Yaskawa INFORM job: OK_R2_O27-28(-60,-90)OKKR.JBI

/JOB
//NAME OK_R2_O27-28(-60,-90)OKKR
///FOLDERNAME X4
//POS
///NPOS 259,259,259,8,0,0
///TOOL 0
///POSTYPE PULSE
///PULSE
C00000=4026,-114538,-112087,-7469,89169,3010
C00001=141886,-58901,-77773,-23947,92184,48931
C00002=141578,-57959,-69842,-23828,88059,49648
C00003=141015,-58362,-68930,-23729,87194,49620
C00004=141015,-58433,-67903,-23734,86579,49742
C00005=141015,-58416,-68203,-23732,86757,49707
C00006=139686,-59077,-68559,-23492,86274,49323
C00007=141015,-58416,-68203,-23732,86757,49707
C00008=141015,-58175,-70675,-23724,88270,49406
C00009=128422,-62662,-73061,-21186,84142,45699
C00010=126942,-63006,-72152,-20876,83082,45360
C00011=125859,-63161,-72230,-20632,82787,45027
C00012=126427,-63083,-72191,-20760,82941,45202
C00013=126427,-63151,-70840,-20793,82126,45342
C00014=126555,-60703,-71087,-20771,83482,45154
C00015=126555,-60807,-69619,-20804,82583,45308
C00016=127911,-60340,-72276,-21054,84679,45425
C00017=126649,-37475,-64724,-20742,91025,43893
C00018=125827,-36059,-63222,-20543,90649,43679
C00019=125029,-36163,-63287,-20349,90451,43443
C00020=125623,-36090,-63238,-20492,90597,43620
C00021=125567,-34509,-61579,-20475,90388,43635
C00022=125623,-36090,-63238,-20492,90597,43620
C00023=136338,-54772,-80020,-22951,93924,46664
C00024=126842,-100836,-98035,7484,62353,-34456
C00025=121554,-58479,-70523,23610,81393,-54658
C00026=122608,-55102,-66306,23365,80313,-54492
C00027=122608,-55177,-65231,23407,79671,-54618
C00028=122608,-55168,-65391,23401,79766,-54599
C00029=123914,-55086,-65345,23053,79422,-54193
C00030=122608,-54831,-68633,23286,81762,-54205
C00031=135057,-52399,-66134,19707,78324,-50392
C00032=136320,-52036,-64863,19353,77466,-50085
C00033=137087,-51720,-64683,19108,77338,-49833
C00034=136456,-51981,-64832,19310,77443,-50041
C00035=136456,-52079,-63836,19355,76815,-50143
C00036=136990,-51767,-64649,19142,77318,-49872
C00037=137022,-51845,-63710,19174,76726,-49958
C00038=136456,-51987,-64775,19313,77407,-50047
C00039=133944,-28024,-57248,19775,85241,-49647
C00040=134132,-26753,-56119,19717,85158,-49597
C00041=134834,-26485,-55932,19497,85022,-49384
C00042=134200,-26728,-56101,19696,85144,-49576
C00043=134114,-25902,-54940,19729,84890,-49647
C00044=134200,-26728,-56101,19696,85144,-49576
C00045=118482,-33028,-63104,24263,90056,-53997
C00046=122367,-92922,-80640,24281,48069,-47816
C00047=126786,-89890,-74695,22151,44886,-46448
C00048=127161,-97737,-79785,22235,43950,-46500
C00049=123248,-90194,-74818,24549,45815,-47997
C00050=127415,-97816,-73172,23855,40088,-47458
C00051=126170,-63328,-70330,17365,77748,-40778
C00052=125190,-29892,-53752,19424,104543,-36953
C00053=126048,-60244,-72015,19024,100224,-37353
C00054=129257,-118219,-89475,18745,55248,-43183
C00055=137691,-142606,-72024,68262,8176,-68089
C00056=133583,-154957,-83359,69355,10840,-69277
C00057=143208,-69932,-76566,3835,55131,-38143
C00058=145269,-69372,-74031,2532,53783,-37349
C00059=145623,-70560,-74318,2309,53334,-37215
C00060=145877,-71977,-74674,2159,52821,-37126
C00061=150479,-88391,-71295,-7827,30676,-34231
C00062=155149,-99562,-68728,-17073,24216,-29422
C00063=155171,-99618,-68748,-17116,24204,-29400
C00064=147593,-80029,-75214,3987,58057,-35963
C00065=135411,-30256,-54215,19906,99237,-39191
C00066=136924,-45266,-63867,20529,99583,-42128
C00067=135919,-63282,-79199,18518,95221,-35974
C00068=132995,-62152,-82050,19008,98077,-36535
C00069=146597,-77867,-86304,-14777,77362,40583
C00070=149051,-83920,-77966,-27962,61330,43366
C00071=147016,-82878,-78861,-27270,61762,42356
C00072=150258,-80090,-74192,-28972,61572,43794
C00073=147203,-82736,-75214,-27895,59886,42937
C00074=149174,-90821,-74362,-30094,56451,44819
C00075=149181,-90838,-74335,-30106,56432,44829
C00076=142127,-55357,-68668,-16008,88190,36417
C00077=139597,-29306,-55135,-13561,105265,43860
C00078=139307,-22183,-50052,-13420,110648,48850
C00079=143000,-50940,-68567,-12955,107923,50473
C00080=151384,-106281,-89249,-20779,70795,55648
C00081=160066,-126367,-88243,-34868,53700,64122
C00082=163396,-129603,-85950,-37116,52558,66246
C00083=170124,-141759,-99198,-37878,56949,67763
C00084=136065,-86573,-88427,-19738,64261,50781
C00085=131238,-34371,-67556,-16142,92767,44746
C00086=129250,-31705,-63617,-15587,92385,44136
C00087=129352,-32707,-64477,-15613,92413,44167
C00088=131697,-69478,-76768,-20363,65108,48613
C00089=131773,-70326,-76955,-20450,64822,48696
C00090=132058,-74122,-77463,-20852,63359,49080
C00091=133339,-88291,-77768,-22923,57086,50905
C00092=133349,-88399,-77812,-22935,57064,50915
C00093=131196,-63810,-72799,-16490,80948,46201
C00094=129177,-28734,-55041,-14328,108045,42506
C00095=130098,-48812,-67542,-14099,105651,43119
C00096=135207,-44513,-73407,-14614,112147,44115
C00097=29949,-45667,-74098,-14599,111934,44036
C00098=58439,-77793,-131196,12526,65130,-72907
C00099=127967,-68734,-129505,14303,77633,-40887
C00100=95610,-66837,-124865,12878,106964,29326
C00101=114477,-82986,-128069,-10037,99362,30876
C00102=114477,-86675,-127599,-9968,97208,31049
C00103=114477,-85869,-127717,-9982,97688,31010
C00104=112971,-85457,-127558,-9480,97652,30583
C00105=92898,-68043,-124184,12345,107279,29217
C00106=94676,-96172,-135168,11342,99536,28957
C00107=94658,-98853,-133311,11256,97065,28724
C00108=95162,-93948,-131570,11149,98431,28996
C00109=94658,-98853,-133311,11256,97065,28724
C00110=98957,-93279,-135892,10098,100972,30314
C00111=110651,-49645,-111382,-11454,101977,41926
C00112=110651,-52306,-111062,-11381,100444,42072
C00113=110651,-51032,-111225,-11415,101184,42001
C00114=109332,-50612,-111005,-10903,101130,41666
C00115=110651,-51032,-111225,-11415,101184,42001
C00116=95349,-81608,-124870,6979,89211,41800
C00117=95569,-84274,-123262,6885,86851,41730
C00118=95987,-80853,-121877,6703,87721,41895
C00119=95620,-84218,-124899,6861,87878,41800
C00120=95569,-64927,-125294,6988,97966,42345
C00121=68892,-69920,-123147,37382,97488,27376
C00122=68892,-69920,-123147,37382,97488,27376
C00123=68031,-90449,-131916,26273,102698,-13010
C00124=71990,-90821,-130319,24971,100628,-12221
C00125=79202,-85723,-129933,18399,102227,-11158
C00126=79202,-87573,-129743,18299,101214,-11319
C00127=79215,-86748,-129802,18348,101647,-11244
C00128=80019,-82599,-128205,18192,102594,-10863
C00129=79215,-83561,-130075,18500,103364,-10977
C00130=72693,-92471,-130926,24716,100020,-12130
C00131=84462,-79485,-128908,14471,105620,-10048
C00132=84462,-81364,-128782,14389,104604,-10171
C00133=84462,-80152,-128866,14442,105265,-10090
C00134=85127,-76283,-127309,14327,106169,-9791
C00135=84083,-80509,-129856,14589,105729,-10142
C00136=72693,-92471,-130926,24716,100020,-12130
C00137=84410,-93585,-133880,14135,99565,-10800
C00138=84410,-96087,-133656,14067,98184,-10958
C00139=84410,-94757,-133784,14102,98923,-10874
C00140=85385,-88254,-131421,13878,100620,-10395
C00141=84410,-93524,-133885,14136,99597,-10796
C00142=71593,-80403,-130713,25764,105804,-11193
C00143=71593,-76518,-130795,32588,107642,-50773
C00144=78737,-74748,-122692,29451,101785,-50195
C00145=78737,-75119,-122640,29424,101590,-50246
C00146=78737,-77656,-122235,29243,100229,-50601
C00147=78737,-76000,-122510,29360,101124,-50368
C00148=80423,-78738,-123652,28717,100035,-50114
C00149=74556,-86649,-127298,30428,100128,-51983
C00150=80828,-115772,-134875,23515,87622,-34169
C00151=81779,-109674,-132899,23210,89145,-33553
C00152=81251,-111521,-134487,23382,89304,-33698
C00153=81251,-105171,-135824,23470,93068,-32958
C00154=68840,-107115,-136272,27319,95724,-36434
C00155=63225,-73448,-121715,35441,110616,-40683
C00156=63225,-75726,-121350,35103,109465,-41078
C00157=63225,-74780,-121511,35242,109948,-40913
C00158=64274,-77370,-122606,34819,109058,-40843
C00159=63225,-72176,-121887,35634,111241,-40463
C00160=49970,-81546,-125790,38107,113825,-44363
///LIMIT ON
C00161=57709,-122397,-137101,29737,92456,-40867
///LIMIT OFF
C00162=58596,-119094,-136084,29567,93103,-40381
///LIMIT ON
C00163=57709,-122397,-137101,29737,92456,-40867
///LIMIT OFF
C00164=55203,-68367,-119401,40200,117926,-44687
C00165=60082,-69241,-118655,38808,115482,-43833
C00166=70586,-91755,-127960,28719,99346,-36878
C00167=58188,-109460,-135678,31383,99168,-40913
C00168=58490,-112528,-136667,30978,97870,1529
C00169=60906,-115834,-135191,27280,87192,7891
C00170=59523,-104900,-131558,29509,92292,6762
C00171=56755,-69637,-113373,48283,106573,15620
C00172=54350,-66602,-110106,52807,107764,16888
C00173=41617,-83627,-112954,60214,104174,10782
C00174=28595,-74588,-109030,64073,112578,9715
C00175=27901,-74856,-109516,64304,113044,9684
C00176=47677,-91044,-131006,33540,104945,-26933
///LIMIT ON
C00177=61912,-123095,-136997,21835,82960,-21144
///LIMIT OFF
C00178=55245,-67359,-115879,41246,114826,-18847
C00179=56373,-63948,-120424,31486,113982,-21878
C00180=60160,-119068,-134198,40501,98040,-56836
C00181=60160,-114231,-136050,40991,100824,-55736
C00182=83270,-65163,-115072,44519,104941,-68495
C00183=85626,-71751,-115611,43145,101762,-69006
C00184=84703,-74765,-113322,46278,99950,-69048
C00185=88262,-57949,-105339,45732,101061,-67072
C00186=101128,-54439,-109788,29647,101331,-67085
C00187=94109,-71359,-120991,32482,95089,-70619
C00188=139920,-94168,-131864,-18457,87392,-68872
C00189=164516,-97279,-127794,-42983,94890,-67354
C00190=173049,-108773,-127338,-48480,95293,-64880
C00191=167455,-99667,-123526,-46768,91665,-65667
C00192=150655,-112829,-124924,-46404,81551,-69570
C00193=121485,-77048,-127419,1615,96838,-70506
C00194=141399,-68559,-121452,-18612,100542,-82408
C00195=124764,-66998,-122517,455,101591,-69580
C00196=125438,-65497,-122047,206,102070,-69406
C00197=126763,-65065,-121637,-284,102041,-69063
C00198=120566,-81356,-130422,1967,92166,-70821
C00199=120566,-76874,-130556,1975,94549,-70784
C00200=125831,-89175,-135984,-584,100456,3377
C00201=135444,-90328,-133818,-3844,98745,6043
C00202=135106,-91582,-131067,-3703,96397,6020
C00203=109572,-93250,-131605,4930,96041,-1221
C00204=87998,-80897,-129766,12221,103039,-6801
C00205=120367,-85836,-132161,9477,101125,-4686
C00206=121843,-84446,-127481,8917,98851,-4443
C00207=141527,-76678,-124327,2331,99777,1071
C00208=129396,-87762,-136435,6506,102049,-2146
C00209=130312,-90929,-132015,6094,97669,-2118
C00210=129363,-86126,-129166,6424,98441,-2343
C00211=154391,-66262,-120817,-2111,102954,4533
C00212=150219,-78004,-128736,-656,101737,3438
C00213=144801,-93164,-134458,-6692,98136,8453
C00214=144714,-84238,-128290,-6682,98918,8387
C00215=123987,-96369,-132727,351,94749,2642
C00216=117273,-90923,-135342,2652,99260,807
C00217=121768,-81824,-133505,6628,103406,-2316
C00218=156634,-61907,-126378,-3075,94108,-72042
C00219=137751,-95208,-134275,-20772,87240,-85897
C00220=160150,-96114,-119425,-47944,88000,-84014
C00221=155632,-76142,-111175,-46420,89477,-86695
C00222=140577,-51697,-109067,-28499,100390,-90208
C00223=132515,-86588,-130828,-12209,89399,-86569
C00224=131433,-65917,-122271,-11801,94519,-87353
C00225=105014,-130347,-135310,35662,68949,-87927
C00226=104111,-122678,-131012,37838,71563,-88295
C00227=106068,-95108,-121457,35727,77495,-85456
C00228=111976,-92342,-121116,28689,76109,-84990
C00229=109886,-91804,-124961,29447,79067,-84948
C00230=149255,-76965,-128804,-12913,97351,-82067
C00231=139576,-84817,-129459,-1876,92119,-81977
C00232=148153,-75159,-124875,-14582,97706,-83124
C00233=147471,-74687,-124680,-14327,97728,-83315
C00234=146233,-76138,-125285,-13834,97200,-83595
C00235=149105,-93032,-135747,-12738,93444,-81701
C00236=185390,-49383,-101810,-59538,112858,-87685
C00237=178512,-86634,-117153,-49673,98332,-85874
C00238=173349,-72532,-111075,-48613,98244,-88135
C00239=168036,-108473,-125463,-40279,80417,-90424
C00240=177281,-105060,-127213,-43325,86617,-89102
C00241=179538,-98194,-126909,-44097,90073,-89650
C00242=186838,-121222,-134600,-46262,88364,-34815
C00243=184942,-111108,-129526,-47770,92446,-34323
C00244=190696,-133181,-128203,-55352,82590,-27191
C00245=183298,-110716,-114958,-62940,86926,-24714
C00246=183340,-79337,-102682,-66907,100105,-26093
C00247=185184,-79882,-104966,-67590,101694,-26340
C00248=200556,-111348,-116827,-65901,96352,-23239
C00249=198058,-141281,-124059,-63896,81460,-21046
C00250=197686,-130606,-120716,-64143,86176,-21704
C00251=190742,-91685,-107319,-68355,104344,-23733
C00252=191763,-88052,-108908,-69399,106084,-24879
C00253=198707,-113921,-124746,-62747,95061,-23584
C00254=198707,-113921,-124746,-62747,95061,-23584
C00255=177230,-52335,-122859,-28636,110825,-71925
C00256=181545,-112898,-119475,-62736,95065,-23495
C00257=7977,-118181,-126139,1257,90741,84078
C00258=4441,-114902,-113556,-6551,89340,11522
BC00000=154724,492605,1071101
BC00001=345701,440224,1074748
BC00002=345701,440224,1074748
BC00003=345701,440224,1074748
BC00004=345701,440224,1074748
BC00005=345701,440224,1074748
BC00006=345701,440224,1074748
BC00007=345701,440224,1074748
BC00008=345701,440224,1074748
BC00009=345701,440224,1074748
BC00010=345701,440224,1074748
BC00011=345701,440224,1074748
BC00012=345701,440224,1074748
BC00013=345701,440224,1074748
BC00014=345701,440224,1074748
BC00015=345701,440224,1074748
BC00016=345701,440224,1074748
BC00017=345701,440224,1074748
BC00018=345701,440224,1074748
BC00019=345701,440224,1074748
BC00020=345701,440224,1074748
BC00021=345701,440224,1074748
BC00022=345701,440224,1074748
BC00023=345701,440224,1074748
BC00024=136420,445856,1074364
BC00025=136420,445856,1074364
BC00026=136419,445855,1074361
BC00027=136419,445855,1074361
BC00028=136419,445855,1074361
BC00029=136419,445855,1074361
BC00030=136419,445855,1074361
BC00031=136419,445855,1074361
BC00032=136419,445855,1074361
BC00033=136419,445855,1074361
BC00034=136419,445855,1074361
BC00035=136419,445855,1074361
BC00036=136419,445855,1074361
BC00037=136419,445855,1074361
BC00038=136419,445855,1074361
BC00039=136419,445855,1074361
BC00040=136419,445855,1074361
BC00041=136419,445855,1074361
BC00042=136419,445855,1074361
BC00043=136419,445855,1074361
BC00044=136419,445855,1074361
BC00045=136419,445855,1074361
BC00046=132124,434884,1075130
BC00047=132124,434884,1075130
BC00048=132124,434884,1075130
BC00049=132124,434884,1075130
BC00050=132125,434884,1075124
BC00051=132124,434884,1075127
BC00052=132124,434884,1075127
BC00053=132124,434884,1075127
BC00054=132124,434884,1075127
BC00055=132124,434884,1075127
BC00056=132124,434884,1075123
BC00057=132124,434884,1075123
BC00058=132124,434884,1075123
BC00059=132124,434884,1075123
BC00060=132124,434884,1075123
BC00061=132124,434884,1075123
BC00062=132124,434884,1075120
BC00063=132124,434884,1075120
BC00064=132124,434884,1075123
BC00065=132124,434884,1075120
BC00066=132124,434884,1075120
BC00067=132124,434884,1075120
BC00068=132124,434884,1075120
BC00069=365171,434884,1075120
BC00070=365171,434884,1075120
BC00071=365171,434884,1075120
BC00072=365171,434884,1075120
BC00073=365171,434884,1075120
BC00074=365171,434884,1075120
BC00075=365171,434884,1075120
BC00076=365171,434884,1075120
BC00077=365171,434884,1075120
BC00078=365171,434884,1075120
BC00079=365171,434884,1075120
BC00080=365171,434884,1075120
BC00081=365171,434884,1075120
BC00082=365171,434884,1075120
BC00083=365171,434884,1075120
BC00084=365171,434884,1075120
BC00085=365171,434884,1075120
BC00086=365171,434884,1075120
BC00087=365171,434884,1075120
BC00088=365171,434884,1075120
BC00089=365171,434884,1075120
BC00090=365171,434884,1075120
BC00091=365171,434884,1075120
BC00092=365171,434884,1075120
BC00093=365171,434884,1075120
BC00094=365171,434884,1075120
BC00095=365171,434884,1075120
BC00096=365171,434884,1075120
BC00097=261029,496377,1070955
BC00098=158954,465505,1070842
BC00099=76268,391428,1075124
BC00100=6523,355122,1075124
BC00101=1090,352294,1075124
BC00102=1090,352294,1075124
BC00103=1090,352294,1075124
BC00104=1090,352294,1075124
BC00105=1090,352294,1075124
BC00106=1090,352294,1075124
BC00107=1090,352294,1075124
BC00108=1090,352294,1075124
BC00109=1090,352294,1075124
BC00110=1090,352294,1075124
BC00111=1090,352294,1075124
BC00112=1090,352294,1075124
BC00113=1090,352294,1075124
BC00114=1090,352294,1075124
BC00115=1090,352294,1075124
BC00116=1090,352294,1075124
BC00117=1090,352294,1075124
BC00118=1090,352294,1075124
BC00119=1090,352294,1075124
BC00120=1090,352294,1075124
BC00121=1090,352294,1075124
BC00122=1090,352294,1075124
BC00123=119522,336763,1061257
BC00124=119522,336763,1061257
BC00125=119522,336763,1061257
BC00126=119523,336764,1061256
BC00127=119522,336763,1061257
BC00128=119522,336763,1061257
BC00129=119522,336763,1061257
BC00130=177823,336763,1064589
BC00131=177823,336763,1061257
BC00132=177823,336763,1061257
BC00133=177823,336763,1061257
BC00134=177823,336763,1061257
BC00135=177823,336763,1061257
BC00136=233759,336763,1064589
BC00137=233759,336315,1058464
BC00138=233759,336315,1058464
BC00139=233759,336315,1058464
BC00140=233758,336315,1058463
BC00141=233759,336315,1058464
BC00142=233759,336315,1059003
BC00143=363339,336315,1059003
BC00144=363339,336315,1059003
BC00145=363339,336315,1059003
BC00146=363339,336315,1059003
BC00147=363339,336315,1059003
BC00148=363339,336315,1059003
BC00149=363339,336315,1059003
BC00150=363339,336315,1059003
BC00151=363339,336315,1059003
BC00152=363339,336315,1059003
BC00153=363339,336315,1059003
BC00154=362736,339076,1059003
BC00155=362465,340315,1059003
BC00156=362465,340315,1059003
BC00157=362465,340315,1059003
BC00158=362465,340315,1059003
BC00159=362465,340315,1059003
BC00160=362465,340315,1059003
BC00161=362465,340315,1059003
BC00162=362465,340315,1059003
BC00163=362465,340315,1059003
BC00164=362465,340315,1059003
BC00165=362465,340315,1059003
BC00166=362465,340315,1059003
BC00167=362465,340315,1059003
BC00168=362466,340316,1059002
BC00169=349813,347319,1059002
BC00170=349813,347319,1059002
BC00171=349813,347319,1059002
BC00172=349813,347319,1059002
BC00173=349813,347319,1059002
BC00174=349813,347319,1059002
BC00175=349813,347319,1059002
BC00176=349813,347319,1059002
BC00177=348803,347319,1059002
BC00178=349813,347319,1059002
BC00179=349813,347319,1059002
BC00180=381408,339179,1066112
BC00181=381408,339179,1066112
BC00182=396370,339179,1066112
BC00183=396370,339179,1066112
BC00184=396370,339179,1066112
BC00185=396370,339179,1066112
BC00186=396370,339179,1066112
BC00187=396370,339179,1066112
BC00188=396370,330317,1066112
BC00189=396370,323887,1066112
BC00190=396370,323887,1066112
BC00191=396370,323887,1066112
BC00192=366417,324055,1066112
BC00193=396370,328332,1066112
BC00194=396370,328332,1066109
BC00195=396370,328332,1066112
BC00196=396370,328332,1066112
BC00197=396370,328332,1066112
BC00198=396370,328332,1066112
BC00199=396370,328332,1066112
BC00200=237361,342916,1066112
BC00201=237361,342915,1066109
BC00202=237361,342915,1066109
BC00203=237361,342915,1066109
BC00204=237361,342915,1066109
BC00205=204586,344800,1071989
BC00206=204586,344800,1071989
BC00207=204586,344800,1071989
BC00208=248457,342915,1066109
BC00209=248457,342915,1066109
BC00210=248457,342915,1066109
BC00211=248457,342915,1066109
BC00212=248457,342915,1066109
BC00213=280970,342915,1066109
BC00214=280970,342915,1066109
BC00215=280970,342915,1066109
BC00216=280970,342915,1066109
BC00217=250684,342915,1066109
BC00218=120387,342915,1066109
BC00219=43564,342915,1066109
BC00220=43564,342915,1066109
BC00221=43564,342915,1066109
BC00222=43564,342915,1066109
BC00223=43563,342915,1066106
BC00224=43563,352075,1066106
BC00225=77352,343027,1066106
BC00226=77352,343027,1066106
BC00227=77352,343027,1066106
BC00228=77352,343027,1066106
BC00229=77352,343027,1066106
BC00230=77352,325808,1066106
BC00231=77351,325808,1066103
BC00232=77352,325808,1066106
BC00233=77352,325808,1066106
BC00234=77352,325808,1066106
BC00235=77352,325808,1066106
BC00236=58352,353191,1066106
BC00237=58352,353191,1066106
BC00238=58352,353191,1066106
BC00239=58352,353191,1066106
BC00240=58352,353191,1066106
BC00241=58352,353191,1066106
BC00242=58352,353191,1066106
BC00243=58352,353191,1066106
BC00244=58352,353191,1066106
BC00245=58352,353191,1066106
BC00246=58352,353191,1066106
BC00247=58352,353191,1066106
BC00248=58352,353191,1066106
BC00249=58352,353191,1066106
BC00250=58352,353191,1066106
BC00251=58352,353191,1066106
BC00252=58352,353191,1066106
BC00253=58352,353191,1066106
BC00254=12917,447675,1066106
BC00255=70552,358579,1066106
BC00256=12917,447675,1066106
BC00257=12917,516869,1066106
BC00258=138844,495152,1070575
EC00000=454111,372643
EC00001=443859,372643
EC00002=443859,372643
EC00003=443859,372643
EC00004=443859,372643
EC00005=443859,372643
EC00006=443859,372643
EC00007=443859,372643
EC00008=443859,372643
EC00009=443859,372643
EC00010=443859,372643
EC00011=443859,372643
EC00012=443859,372643
EC00013=443859,372643
EC00014=443859,372643
EC00015=443859,372643
EC00016=443859,372643
EC00017=443859,372643
EC00018=443859,372643
EC00019=443859,372643
EC00020=443859,372643
EC00021=443859,372643
EC00022=443859,372643
EC00023=443859,372643
EC00024=444967,372643
EC00025=444967,372643
EC00026=444965,372643
EC00027=444965,372643
EC00028=444965,372643
EC00029=444965,372643
EC00030=444965,372643
EC00031=444965,372643
EC00032=444965,372643
EC00033=444965,372643
EC00034=444965,372643
EC00035=444965,372643
EC00036=444965,372643
EC00037=444965,372643
EC00038=444965,372643
EC00039=444965,372643
EC00040=444965,372643
EC00041=444965,372643
EC00042=444965,372643
EC00043=444965,372643
EC00044=444965,372643
EC00045=444965,372643
EC00046=442821,372643
EC00047=442821,372643
EC00048=442821,372643
EC00049=442821,372643
EC00050=442817,372643
EC00051=442818,372643
EC00052=442818,372643
EC00053=442818,372643
EC00054=442818,372643
EC00055=442818,372643
EC00056=442816,372643
EC00057=442816,372643
EC00058=442816,372643
EC00059=442816,372643
EC00060=442816,372643
EC00061=442816,372643
EC00062=442815,372643
EC00063=442815,372643
EC00064=442816,372643
EC00065=442814,372643
EC00066=442814,372643
EC00067=442814,372643
EC00068=442814,372643
EC00069=442814,372643
EC00070=442814,372643
EC00071=442814,372643
EC00072=442814,372643
EC00073=442814,372643
EC00074=442814,372643
EC00075=442814,372643
EC00076=442814,372643
EC00077=442814,372643
EC00078=442814,372643
EC00079=442814,372643
EC00080=442814,372643
EC00081=442814,372643
EC00082=442814,372643
EC00083=442814,372643
EC00084=442814,372643
EC00085=442814,372643
EC00086=442814,372643
EC00087=442814,372643
EC00088=442814,372643
EC00089=442814,372643
EC00090=442814,372643
EC00091=442814,372643
EC00092=442814,372643
EC00093=442814,372643
EC00094=442814,372643
EC00095=442814,372643
EC00096=442814,372643
EC00097=442814,372643
EC00098=798155,372644
EC00099=798157,372644
EC00100=798157,372644
EC00101=798157,372644
EC00102=798157,372644
EC00103=798157,372644
EC00104=798157,372644
EC00105=798157,372644
EC00106=798157,372644
EC00107=798157,372644
EC00108=798157,372644
EC00109=798157,372644
EC00110=798157,372644
EC00111=798157,372644
EC00112=798157,372644
EC00113=798157,372644
EC00114=798157,372644
EC00115=798157,372644
EC00116=798157,372644
EC00117=798157,372644
EC00118=798157,372644
EC00119=798157,372644
EC00120=798157,372644
EC00121=798157,372644
EC00122=798157,372644
EC00123=798157,372644
EC00124=798157,372644
EC00125=798157,372644
EC00126=798156,372644
EC00127=798157,372644
EC00128=798157,372644
EC00129=798157,372644
EC00130=798157,372644
EC00131=798157,372644
EC00132=798157,372644
EC00133=798157,372644
EC00134=798157,372644
EC00135=798157,372644
EC00136=798157,372644
EC00137=798157,372644
EC00138=798157,372644
EC00139=798157,372644
EC00140=798155,372644
EC00141=798157,372644
EC00142=798157,372644
EC00143=798157,372644
EC00144=798157,372644
EC00145=798157,372644
EC00146=798157,372644
EC00147=798157,372644
EC00148=798157,372644
EC00149=798157,372644
EC00150=798157,372644
EC00151=798157,372644
EC00152=798157,372644
EC00153=798157,372644
EC00154=798157,372644
EC00155=798157,372644
EC00156=798157,372644
EC00157=798157,372644
EC00158=798157,372644
EC00159=798157,372644
EC00160=798157,372644
EC00161=798157,372644
EC00162=798157,372644
EC00163=798157,372644
EC00164=798157,372644
EC00165=798157,372644
EC00166=798157,372644
EC00167=798157,372644
EC00168=798156,372644
EC00169=798156,372644
EC00170=798156,372644
EC00171=798156,372644
EC00172=798156,372644
EC00173=798156,372644
EC00174=798156,372644
EC00175=798156,372644
EC00176=798156,372644
EC00177=798156,372644
EC00178=798156,372644
EC00179=798156,372644
EC00180=798156,372644
EC00181=798156,372644
EC00182=798156,372644
EC00183=798156,372644
EC00184=798156,372644
EC00185=798156,372644
EC00186=798156,372644
EC00187=798156,372644
EC00188=798156,372644
EC00189=798156,372644
EC00190=798156,372644
EC00191=798156,372644
EC00192=798156,372644
EC00193=798156,372644
EC00194=798155,372645
EC00195=798156,372644
EC00196=798156,372644
EC00197=798156,372644
EC00198=798156,372644
EC00199=798156,372644
EC00200=798156,372644
EC00201=798155,372644
EC00202=798155,372644
EC00203=798155,372644
EC00204=798155,372644
EC00205=798155,372644
EC00206=798155,372644
EC00207=798155,372644
EC00208=798155,372644
EC00209=798155,372644
EC00210=798155,372644
EC00211=798155,372644
EC00212=798155,372644
EC00213=798155,372644
EC00214=798155,372644
EC00215=798155,372644
EC00216=798155,372644
EC00217=798155,372644
EC00218=798155,372644
EC00219=798155,372644
EC00220=798155,372644
EC00221=798155,372644
EC00222=798155,372644
EC00223=798154,372644
EC00224=798154,372644
EC00225=798154,372644
EC00226=798154,372644
EC00227=798154,372644
EC00228=798154,372644
EC00229=798154,372644
EC00230=798154,372644
EC00231=798152,372644
EC00232=798154,372644
EC00233=798154,372644
EC00234=798154,372644
EC00235=798154,372644
EC00236=798154,372644
EC00237=798154,372644
EC00238=798154,372644
EC00239=798154,372644
EC00240=798154,372644
EC00241=798154,372644
EC00242=798154,372644
EC00243=798154,372644
EC00244=798154,372644
EC00245=798154,372644
EC00246=798154,372644
EC00247=798154,372644
EC00248=798154,372644
EC00249=798154,372644
EC00250=798154,372644
EC00251=798154,372644
EC00252=798154,372644
EC00253=798154,372644
EC00254=798154,372644
EC00255=798154,372644
EC00256=798154,372644
EC00257=798154,372644
EC00258=0,372643
///POSTYPE BASE
///RECTAN
///RCONF 0,0,0,0,1,0,0,0,0,0,0,0,0,0,0,0,0,0,0,0,0,0,0,0
P00006=2.006,1.622,-0.565,0.0000,0.0000,0.0000
P00021=0.073,2.058,-0.109,0.0000,0.0000,0.0000
P00022=2.006,1.622,-0.565,0.0000,0.0000,0.0000
///RCONF 0,0,0,0,0,0,0,0,0,0,0,0,0,0,0,0,0,0,0,0,0,0,0,0
P00023=-2.957,-4.083,2.762,0.0000,0.0000,0.0000
P00024=-1.466,-0.226,-0.419,0.0000,0.0000,0.0000
P00025=3.643,0.007,-2.585,0.0000,0.0000,0.0000
P00026=2.644,0.055,-2.583,0.0000,0.0000,0.0000
P00027=2.278,0.099,-4.210,0.0000,0.0000,0.0000
//INST
///DATE 2024/11/18 14:52
///ATTR SC,RW
///GROUP1 RB1,BS1
///GROUP2 ST1
NOP
SFTOF3D
'NOWY PROGRAM KM
SFTOF3D
MOVJ C00000 BC00000 VJ=100.00  +MOVJ EC00000 VJ=100.00
'POMIAR
MOVJ C00001 BC00001 VJ=100.00  +MOVJ EC00001 VJ=100.00
MOVJ C00002 BC00002 VJ=100.00  +MOVJ EC00002 VJ=100.00
SMOVL C00003 BC00003 V=100.0  +MOVJ EC00003
SREFP 3 C00004 BC00004  +REFP EC00004
CALL JOB:SEARCH-R1-S13D
SET P024 P006
SFTON3D P024
SMOVL C00005 BC00005 V=100.0  +MOVJ EC00005
SREFP 3 C00006 BC00006  +REFP EC00006
CALL JOB:SEARCH-R1-S13D
SET P024 P006
SFTON3D P024
SFTOF3D
SMOVL C00007 BC00007 V=166.7  +MOVJ EC00007
MOVJ C00008 BC00008 VJ=100.00  +MOVJ EC00008 VJ=100.00
MOVJ C00009 BC00009 VJ=100.00  +MOVJ EC00009 VJ=100.00
SMOVL C00010 BC00010 V=100.0  +MOVJ EC00010
SREFP 3 C00011 BC00011  +REFP EC00011
CALL JOB:SEARCH-R1-S13D
SET P025 P006
SFTON3D P025
SMOVL C00012 BC00012 V=100.0  +MOVJ EC00012
SREFP 3 C00013 BC00013  +REFP EC00013
CALL JOB:SEARCH-R1-S13D
SET P025 P006
SFTON3D P025
SFTOF3D
SMOVL C00014 BC00014 V=166.7  +MOVJ EC00014
SREFP 3 C00015 BC00015  +REFP EC00015
CALL JOB:SEARCH-R1-S13D
SET P026 P006
SFTON3D P026
SMOVL C00016 BC00016 V=250.0  +MOVJ EC00016
SMOVL C00017 BC00017 V=400.0  +MOVJ EC00017
SMOVL C00018 BC00018 V=100.0  +MOVJ EC00018
SREFP 3 C00019 BC00019  +REFP EC00019
CALL JOB:SEARCH-R1-S13D
SET P026 P006
SFTON3D P026
SMOVL C00020 BC00020 V=100.0  +MOVJ EC00020
SREFP 3 C00021 BC00021  +REFP EC00021
CALL JOB:SEARCH-R1-S13D
SET P026 P006
SFTON3D P026
SMOVL C00022 BC00022 V=166.7  +MOVJ EC00022
MOVJ C00023 BC00023 VJ=100.00  +MOVJ EC00023 VJ=100.00
MOVJ C00024 BC00024 VJ=100.00  +MOVJ EC00024 VJ=100.00
MOVJ C00025 BC00025 VJ=100.00  +MOVJ EC00025 VJ=100.00
SMOVL C00026 BC00026 V=100.0  +MOVJ EC00026
SREFP 3 C00027 BC00027  +REFP EC00027
CALL JOB:SEARCH-R1-S13D
SET P021 P006
SFTON3D P021
SMOVL C00028 BC00028 V=100.0  +MOVJ EC00028
SREFP 3 C00029 BC00029  +REFP EC00029
CALL JOB:SEARCH-R1-S13D
SET P021 P006
SFTON3D P021
SMOVL C00030 BC00030 V=166.7  +MOVJ EC00030
SMOVL C00031 BC00031 V=416.7  +MOVJ EC00031
SMOVL C00032 BC00032 V=100.0  +MOVJ EC00032
SREFP 3 C00033 BC00033  +REFP EC00033
CALL JOB:SEARCH-R1-S13D
SET P021 P006
SFTON3D P021
SMOVL C00034 BC00034 V=100.0  +MOVJ EC00034
SREFP 3 C00035 BC00035  +REFP EC00035
CALL JOB:SEARCH-R1-S13D
SET P021 P006
SFTON3D P021
SFTOF3D
SMOVL C00036 BC00036 V=166.7  +MOVJ EC00036
SREFP 3 C00037 BC00037  +REFP EC00037
CALL JOB:SEARCH-R1-S13D
SET P022 P006
SFTON3D P022
SMOVL C00038 BC00038 V=166.7  +MOVJ EC00038
SMOVL C00039 BC00039 V=416.7  +MOVJ EC00039
SMOVL C00040 BC00040 V=166.7  +MOVJ EC00040
SREFP 3 C00041 BC00041  +REFP EC00041
CALL JOB:SEARCH-R1-S13D
SET P022 P006
SFTON3D P022
SMOVL C00042 BC00042 V=166.7  +MOVJ EC00042
SREFP 3 C00043 BC00043  +REFP EC00043
CALL JOB:SEARCH-R1-S13D
SET P022 P006
SFTON3D P022
SMOVL C00044 BC00044 V=166.7  +MOVJ EC00044
SMOVL C00045 BC00045 V=666.7  +MOVJ EC00045
SFTOF3D
MOVJ C00046 BC00046 VJ=100.00  +MOVJ EC00046 VJ=100.00
MACRO1 MJ#(0) ARGF9
SFTON3D P021
SMOVL C00047 BC00047 V=166.7  +MOVJ EC00047
SREFP 1 C00048 BC00048  +REFP EC00048
SREFP 2 C00049 BC00049  +REFP EC00049
ARCON
SWVON WEV#(13)
SMOVL C00050 BC00050 V=10.0  +MOVJ EC00050
SMOVL C00051 BC00051 V=10.0  +MOVJ EC00051
SMOVL C00052 BC00052 V=8.3  +MOVJ EC00052
SMOVL C00053 BC00053 V=8.3  +MOVJ EC00053
SMOVL C00054 BC00054 V=8.3  +MOVJ EC00054
SMOVL C00055 BC00055 V=10.0  +MOVJ EC00055
ARCOF
SWVOF
SFTOF3D
SMOVL C00056 BC00056 V=250.0  +MOVJ EC00056
SMOVL C00057 BC00057 V=1000.0  +MOVJ EC00057
MACRO1 MJ#(0) ARGF17
SFTON3D P022
SMOVL C00058 BC00058 V=166.7  +MOVJ EC00058
ARCON
SMOVL C00059 BC00059 V=10.0  +MOVJ EC00059
SMOVL C00060 BC00060 V=10.0  +MOVJ EC00060
SMOVL C00061 BC00061 V=9.2  +MOVJ EC00061
SMOVL C00062 BC00062 V=9.2  +MOVJ EC00062
SMOVC C00063 BC00063 V=9.2  +MOVJ EC00063
SMOVC C00064 BC00064 V=9.2  +MOVJ EC00064
SFTON3D P022
SMOVC C00065 BC00065 V=9.2  +MOVJ EC00065
SMOVL C00066 BC00066 V=9.2  +MOVJ EC00066
ARCOF
SMOVL C00067 BC00067 V=166.7  +MOVJ EC00067
SFTOF3D
MOVJ C00068 BC00068 VJ=100.00  +MOVJ EC00068 VJ=100.00
MOVJ C00069 BC00069 VJ=100.00  +MOVJ EC00069 VJ=100.00
MACRO1 MJ#(0) ARGF9
MOVJ C00070 BC00070 VJ=100.00  +MOVJ EC00070 VJ=100.00
SWVON WEV#(13)
SREFP 1 C00071 BC00071  +REFP EC00071
SREFP 2 C00072 BC00072  +REFP EC00072
SFTON3D P024
SMOVL C00073 BC00073 V=166.7  +MOVJ EC00073
ARCON
SMOVL C00074 BC00074 V=10.0  +MOVJ EC00074
SMOVC C00075 BC00075 V=10.0  +MOVJ EC00075
SMOVC C00076 BC00076 V=10.0  +MOVJ EC00076
SMOVC C00077 BC00077 V=10.0  +MOVJ EC00077
SMOVL C00078 BC00078 V=10.0  +MOVJ EC00078
SMOVL C00079 BC00079 V=10.0  +MOVJ EC00079
SMOVL C00080 BC00080 V=10.0  +MOVJ EC00080
SMOVL C00081 BC00081 V=10.0  +MOVJ EC00081
SMOVL C00082 BC00082 V=10.0  +MOVJ EC00082
ARCOF
SWVOF
SMOVL C00083 BC00083 V=400.0  +MOVJ EC00083
SMOVL C00084 BC00084 V=1000.0  +MOVJ EC00084
SMOVL C00085 BC00085 V=1000.0  +MOVJ EC00085
MACRO1 MJ#(0) ARGF17
SFTON3D P026
SMOVL C00086 BC00086 V=166.7  +MOVJ EC00086
ARCON
SMOVL C00087 BC00087 V=9.2  +MOVJ EC00087
SMOVL C00088 BC00088 V=9.2  +MOVJ EC00088
SMOVL C00089 BC00089 V=9.2  +MOVJ EC00089
SMOVL C00090 BC00090 V=9.2  +MOVJ EC00090
SMOVL C00091 BC00091 V=9.2  +MOVJ EC00091
SMOVC C00092 BC00092 V=9.2  +MOVJ EC00092
SMOVC C00093 BC00093 V=9.2  +MOVJ EC00093
SFTON3D P025
SMOVC C00094 BC00094 V=9.2  +MOVJ EC00094
SMOVL C00095 BC00095 V=8.3  +MOVJ EC00095
ARCOF
SFTOF3D
SMOVL C00096 BC00096 V=250.0  +MOVJ EC00096
MOVJ C00097 BC00097 VJ=100.00  +MOVJ EC00097 VJ=100.00
MACRO1 MJ#(0) ARGF8
'DRUGA POZYCJA
CALL JOB:CLEAN-R1_KM_NEW
MOVJ C00098 BC00098 VJ=100.00  +MOVJ EC00098 VJ=100.00
MOVJ C00099 BC00099 VJ=100.00  +MOVJ EC00099 VJ=20.00
MOVJ C00100 BC00100 VJ=100.00  +MOVJ EC00100 VJ=100.00
'POMIAR
SMOVL C00101 BC00101 V=100.0  +MOVJ EC00101
SREFP 3 C00102 BC00102  +REFP EC00102
CALL JOB:SEARCH-R1-S13D
SET P021 P006
SFTON3D P021
SMOVL C00103 BC00103 V=100.0  +MOVJ EC00103
SREFP 3 C00104 BC00104  +REFP EC00104
CALL JOB:SEARCH-R1-S13D
SET P021 P006
SFTON3D P021
SMOVL C00105 BC00105 V=100.0  +MOVJ EC00105
SMOVL C00106 BC00106 V=100.0  +MOVJ EC00106
SMOVL C00107 BC00107 V=100.0  +MOVJ EC00107
SREFP 3 C00108 BC00108  +REFP EC00108
CALL JOB:SEARCH-R1-S13D
SET P021 P006
SFTON3D P021
SFTOF3D
SMOVL C00109 BC00109 V=100.0  +MOVJ EC00109
SMOVL C00110 BC00110 V=100.0  +MOVJ EC00110
'POMIAR2
SMOVL C00111 BC00111 V=100.0  +MOVJ EC00111
SREFP 3 C00112 BC00112  +REFP EC00112
CALL JOB:SEARCH-R1-S13D
SET P022 P006
SFTON3D P022
SMOVL C00113 BC00113 V=100.0  +MOVJ EC00113
SREFP 3 C00114 BC00114  +REFP EC00114
CALL JOB:SEARCH-R1-S13D
SET P022 P006
SFTON3D P022
SMOVL C00115 BC00115 V=100.0  +MOVJ EC00115
SMOVL C00116 BC00116 V=100.0  +MOVJ EC00116
SMOVL C00117 BC00117 V=100.0  +MOVJ EC00117
SREFP 3 C00118 BC00118  +REFP EC00118
CALL JOB:SEARCH-R1-S13D
SET P022 P006
SFTON3D P022
SFTOF3D
SMOVL C00119 BC00119 V=100.0  +MOVJ EC00119
SMOVL C00120 BC00120 V=100.0  +MOVJ EC00120
SMOVL C00121 BC00121 V=100.0  +MOVJ EC00121
MOVJ C00122 BC00122 VJ=20.00  +MOVJ EC00122 VJ=20.00
MOVJ C00123 BC00123 VJ=50.00  +MOVJ EC00123 VJ=20.00
SMOVL C00124 BC00124 V=100.0  +MOVJ EC00124
'POMIAR3
SMOVL C00125 BC00125 V=100.0  +MOVJ EC00125
SREFP 3 C00126 BC00126  +REFP EC00126
CALL JOB:SEARCH-R1-S13D
SET P023 P006
SFTON3D P023
SMOVL C00127 BC00127 V=100.0  +MOVJ EC00127
SREFP 3 C00128 BC00128  +REFP EC00128
CALL JOB:SEARCH-R1-S13D
SET P023 P006
SFTON3D P023
SMOVL C00129 BC00129 V=100.0  +MOVJ EC00129
'POMIAR4
MOVJ C00130 BC00130 VJ=50.00  +MOVJ EC00130 VJ=20.00
SMOVL C00131 BC00131 V=100.0  +MOVJ EC00131
SREFP 3 C00132 BC00132  +REFP EC00132
CALL JOB:SEARCH-R1-S13D
SET P024 P006
SFTON3D P024
SMOVL C00133 BC00133 V=100.0  +MOVJ EC00133
SREFP 3 C00134 BC00134  +REFP EC00134
CALL JOB:SEARCH-R1-S13D
SET P024 P006
SFTON3D P024
SMOVL C00135 BC00135 V=100.0  +MOVJ EC00135
SFTOF3D
'POMIAR5
MOVJ C00136 BC00136 VJ=50.00  +MOVJ EC00136 VJ=20.00
SMOVL C00137 BC00137 V=100.0  +MOVJ EC00137
SREFP 3 C00138 BC00138  +REFP EC00138
CALL JOB:SEARCH-R1-S13D
SET P025 P006
SFTON3D P025
SMOVL C00139 BC00139 V=100.0  +MOVJ EC00139
SREFP 3 C00140 BC00140  +REFP EC00140
CALL JOB:SEARCH-R1-S13D
SET P025 P006
SFTON3D P025
SMOVL C00141 BC00141 V=100.0  +MOVJ EC00141
SMOVL C00142 BC00142 V=250.0  +MOVJ EC00142
MOVJ C00143 BC00143 VJ=50.00  +MOVJ EC00143 VJ=20.00
SMOVL C00144 BC00144 V=250.0  +MOVJ EC00144
SFTOF3D
'POMIAR6
SMOVL C00145 BC00145 V=100.0  +MOVJ EC00145
SREFP 3 C00146 BC00146  +REFP EC00146
CALL JOB:SEARCH-R1-S13D
SET P026 P006
SFTON3D P026
SMOVL C00147 BC00147 V=100.0  +MOVJ EC00147
SREFP 3 C00148 BC00148  +REFP EC00148
CALL JOB:SEARCH-R1-S13D
SET P026 P006
SFTON3D P026
SMOVL C00149 BC00149 V=100.0  +MOVJ EC00149
SMOVL C00150 BC00150 V=100.0  +MOVJ EC00150
SREFP 3 C00151 BC00151  +REFP EC00151
CALL JOB:SEARCH-R1-S13D
SET P026 P006
SFTON3D P026
SMOVL C00152 BC00152 V=100.0  +MOVJ EC00152
SMOVL C00153 BC00153 V=166.7  +MOVJ EC00153
JUMP *tr
SMOVL C00154 BC00154 V=166.7  +MOVJ EC00154
SFTOF3D
'POMIAR7
SMOVL C00155 BC00155 V=100.0  +MOVJ EC00155
SREFP 3 C00156 BC00156  +REFP EC00156
CALL JOB:SEARCH-R1-S13D
SET P027 P006
SFTON3D P027
SMOVL C00157 BC00157 V=100.0  +MOVJ EC00157
SREFP 3 C00158 BC00158  +REFP EC00158
CALL JOB:SEARCH-R1-S13D
SET P027 P006
SFTON3D P027
SMOVL C00159 BC00159 V=100.0  +MOVJ EC00159
SMOVL C00160 BC00160 V=133.3  +MOVJ EC00160
SMOVL C00161 BC00161 V=100.0  +MOVJ EC00161
SREFP 3 C00162 BC00162  +REFP EC00162
CALL JOB:SEARCH-R1-S13D
SET P027 P006
SFTON3D P027
SMOVL C00163 BC00163 V=100.0  +MOVJ EC00163
SFTOF3D
'SPAWANIE
MACRO1 MJ#(0) ARGF6
SMOVL C00164 BC00164 V=166.7  +MOVJ EC00164
SFTON3D P027
SMOVL C00165 BC00165 V=133.3  +MOVJ EC00165
ARCON
SMOVL C00166 BC00166 V=8.3  +MOVJ EC00166
ARCOF
SMOVL C00167 BC00167 V=166.7  +MOVJ EC00167
SMOVL C00168 BC00168 V=166.7  +MOVJ EC00168
SMOVL C00169 BC00169 V=166.7  +MOVJ EC00169
ARCON
SMOVL C00170 BC00170 V=8.3  +MOVJ EC00170
SMOVL C00171 BC00171 V=8.3  +MOVJ EC00171
SMOVL C00172 BC00172 V=8.3  +MOVJ EC00172
ARCOF
SMOVL C00173 BC00173 V=166.7  +MOVJ EC00173
SMOVL C00174 BC00174 V=166.7  +MOVJ EC00174
MOVJ C00175 BC00175 VJ=20.00  +MOVJ EC00175 VJ=20.00
MOVJ C00176 BC00176 VJ=40.00  +MOVJ EC00176 VJ=20.00
MACRO1 MJ#(0) ARGF6
SMOVL C00177 BC00177 V=133.3  +MOVJ EC00177
ARCON
SMOVL C00178 BC00178 V=13.3  +MOVJ EC00178
ARCOF
SFTOF3D
SMOVL C00179 BC00179 V=166.7  +MOVJ EC00179
SMOVL C00180 BC00180 V=333.3  +MOVJ EC00180
MOVJ C00181 BC00181 VJ=100.00  +MOVJ EC00181 VJ=20.00
*tr
MOVJ C00182 BC00182 VJ=100.00  +MOVJ EC00182 VJ=20.00
SMOVL C00183 BC00183 V=183.3  +MOVJ EC00183
SFTON3D P026
MACRO1 MJ#(0) ARGF21
SMOVL C00184 BC00184 V=133.3  +MOVJ EC00184
ARCON
SMOVL C00185 BC00185 V=10.0  +MOVJ EC00185
SMOVL C00186 BC00186 V=10.0  +MOVJ EC00186
ARCOF
SMOVL C00187 BC00187 V=250.0  +MOVJ EC00187
SMOVL C00188 BC00188 V=250.0  +MOVJ EC00188
SMOVL C00189 BC00189 V=250.0  +MOVJ EC00189
SFTON3D P026
SMOVL C00190 BC00190 V=133.3  +MOVJ EC00190
ARCON
SMOVL C00191 BC00191 V=9.2  +MOVJ EC00191
SMOVL C00192 BC00192 V=10.0  +MOVJ EC00192
ARCOF
SMOVL C00193 BC00193 V=83.3  +MOVJ EC00193
SFTON3D P026
SMOVL C00194 BC00194 V=83.3  +MOVJ EC00194
ARCON
SWVON WEV#(103)
SMOVL C00195 BC00195 V=8.3  +MOVJ EC00195
SMOVL C00196 BC00196 V=9.2  +MOVJ EC00196
SMOVL C00197 BC00197 V=9.2  +MOVJ EC00197
ARCOF
SWVOF
SFTOF3D
SMOVL C00198 BC00198 V=250.0  +MOVJ EC00198
MOVJ C00199 BC00199 VJ=100.00  +MOVJ EC00199 VJ=20.00
MOVJ C00200 BC00200 VJ=80.00  +MOVJ EC00200 VJ=20.00
MOVJ C00201 BC00201 VJ=80.00  +MOVJ EC00201 VJ=20.00
MACRO1 MJ#(0) ARGF14
SFTON3D P024
SMOVL C00202 BC00202 V=166.7  +MOVJ EC00202
ARCON
SMOVL C00203 BC00203 V=11.2  +MOVJ EC00203
ARCOF
SFTOF3D
SMOVL C00204 BC00204 V=250.0  +MOVJ EC00204
SMOVL C00205 BC00205 V=416.7  +MOVJ EC00205
SFTON3D P023
MACRO1 MJ#(0) ARGF14
SMOVL C00206 BC00206 V=133.3  +MOVJ EC00206
ARCON
SMOVL C00207 BC00207 V=10.8  +MOVJ EC00207
ARCOF
SFTOF3D
SMOVL C00208 BC00208 V=250.0  +MOVJ EC00208
SMOVL C00209 BC00209 V=166.7  +MOVJ EC00209
SFTON3D P024
SMOVL C00210 BC00210 V=166.7  +MOVJ EC00210
ARCON
SMOVL C00211 BC00211 V=10.8  +MOVJ EC00211
ARCOF
SFTOF3D
SMOVL C00212 BC00212 V=200.0  +MOVJ EC00212
SMOVL C00213 BC00213 V=416.7  +MOVJ EC00213
SFTON3D P025
SMOVL C00214 BC00214 V=133.3  +MOVJ EC00214
ARCON
SMOVL C00215 BC00215 V=10.8  +MOVJ EC00215
ARCOF
SFTOF3D
SMOVL C00216 BC00216 V=166.7  +MOVJ EC00216
MOVJ C00217 BC00217 VJ=100.00  +MOVJ EC00217 VJ=20.00
MOVJ C00218 BC00218 VJ=100.00  +MOVJ EC00218 VJ=20.00
MOVJ C00219 BC00219 VJ=100.00  +MOVJ EC00219 VJ=20.00
MACRO1 MJ#(0) ARGF21
SFTON3D P022
SMOVL C00220 BC00220 V=250.0  +MOVJ EC00220
ARCON
SMOVL C00221 BC00221 V=9.2  +MOVJ EC00221
SMOVL C00222 BC00222 V=10.0  +MOVJ EC00222
ARCOF
SMOVL C00223 BC00223 V=200.0  +MOVJ EC00223
SMOVL C00224 BC00224 V=166.7  +MOVJ EC00224
SMOVL C00225 BC00225 V=166.7  +MOVJ EC00225
SMOVL C00226 BC00226 V=133.3  +MOVJ EC00226
ARCON
SMOVL C00227 BC00227 V=9.2  +MOVJ EC00227
SMOVL C00228 BC00228 V=10.0  +MOVJ EC00228
ARCOF
SMOVL C00229 BC00229 V=166.7  +MOVJ EC00229
SMOVL C00230 BC00230 V=166.7  +MOVJ EC00230
SMOVL C00231 BC00231 V=133.3  +MOVJ EC00231
ARCON
SWVON WEV#(103)
SMOVL C00232 BC00232 V=8.3  +MOVJ EC00232
SMOVL C00233 BC00233 V=9.2  +MOVJ EC00233
SMOVL C00234 BC00234 V=9.2  +MOVJ EC00234
ARCOF
SWVOF
SMOVL C00235 BC00235 V=166.7  +MOVJ EC00235
JUMP *tro
SMOVL C00236 BC00236 V=166.7  +MOVJ EC00236
MACRO1 MJ#(0) ARGF6
SFTON3D P021
SMOVL C00237 BC00237 V=133.3  +MOVJ EC00237
ARCON
SMOVL C00238 BC00238 V=8.3  +MOVJ EC00238
SMOVL C00239 BC00239 V=8.3  +MOVJ EC00239
ARCOF
SMOVL C00240 BC00240 V=133.3  +MOVJ EC00240
MOVJ C00241 BC00241 VJ=20.00  +MOVJ EC00241 VJ=20.00
MOVJ C00242 BC00242 VJ=100.00  +MOVJ EC00242 VJ=20.00
MOVJ C00243 BC00243 VJ=100.00  +MOVJ EC00243 VJ=20.00
SMOVL C00244 BC00244 V=66.7  +MOVJ EC00244
ARCON
SMOVL C00245 BC00245 V=8.3  +MOVJ EC00245
SMOVL C00246 BC00246 V=8.3  +MOVJ EC00246
ARCOF
MOVJ C00247 BC00247 VJ=20.00  +MOVJ EC00247 VJ=20.00
MOVJ C00248 BC00248 VJ=100.00  +MOVJ EC00248 VJ=20.00
MACRO1 MJ#(0) ARGF6
SMOVL C00249 BC00249 V=100.0  +MOVJ EC00249
ARCON
SMOVL C00250 BC00250 V=13.3  +MOVJ EC00250
SMOVL C00251 BC00251 V=13.3  +MOVJ EC00251
ARCOF
SFTOF3D
SMOVL C00252 BC00252 V=166.7  +MOVJ EC00252
SMOVL C00253 BC00253 V=250.0  +MOVJ EC00253
SMOVL C00254 BC00254 V=1000.0  +MOVJ EC00254
*tro
MOVJ C00255 BC00255 VJ=20.00  +MOVJ EC00255 VJ=20.00
MOVJ C00256 BC00256 VJ=100.00  +MOVJ EC00256 VJ=100.00
MOVJ C00257 BC00257 VJ=100.00  +MOVJ EC00257 VJ=20.00
MOVJ C00258 BC00258 VJ=100.00  +MOVJ EC00258 VJ=100.00
SSFTOF
SFTOF3D
END
